// TIA Portal project "Semafoare_2026" (V15.1)

(* hardware
DEVICE "S71500/ET200MP station_1"  S7-1500 station
   slot 0: "Rail_0"  Rack  6ES7 590-1***0-0AA0
   slot 1: "PLC_1"  CPU 1513-1 PN  6ES7 513-1AL02-0AB0  V2.6
      slot 3: "CPU display_1"  6ES7591-1AA00-0AA0
DEVICE "HMI_1"  KTP900 Basic PN
   slot 0: "HMI_1"  KTP900 Basic PN  6AV2 123-2JB03-0AX0  15.1.0.0
   slot 1: "HMI_RT_1"  KTP900 Basic PN  6AV2 123-2JB03-0AX0  15.1.0.0
   slot 5: "HMI_1.IE_CP_1"  PROFINET Interface  15.0.1.0
      slot 1: "PROFINET Interface_1"  PROFINET Interface
         slot 1: "Port_1"  Port
*)

// ===== PLC "PLC_1"  CPU 1513-1 PN =====

VAR_GLOBAL   // PLC tag table "Default tag table"
   "Clock_Byte" AT %MB0 : Byte;
   "Clock_10Hz" AT %M0.0 : Bool;
   "Clock_5Hz" AT %M0.1 : Bool;
   "Clock_2.5Hz" AT %M0.2 : Bool;
   "Clock_2Hz" AT %M0.3 : Bool;
   "Clock_1.25Hz" AT %M0.4 : Bool;
   "Clock_1Hz" AT %M0.5 : Bool;
   "Clock_0.625Hz" AT %M0.6 : Bool;
   "Clock_0.5Hz" AT %M0.7 : Bool;
END_VAR

DATA_BLOCK "Semafor_masini_ciclu_DB"   // DB1
{ S7_Optimized_Access := 'TRUE' }
VERSION : 0.1
   VAR
      rosu_on : Bool;
      galben_on : Bool;
      galben_on_hmi : Bool;
      verde_on : Bool;
      time_elapsed_rosu : Time;
      time_elapsed_rosu_secunde : Time;
      time_elapsed_verde : Time;
      time_elapsed_verde_secunde : Time;
      time_elapsed_galben : Time;
      time_elapsed_galben_secunde : Time;
      "mod" : Int;
   END_VAR
BEGIN
END_DATA_BLOCK

DATA_BLOCK "Semafor_pietoni_DB"   // DB2
{ S7_Optimized_Access := 'TRUE' }
VERSION : 0.1
BEGIN
END_DATA_BLOCK

DATA_BLOCK "Semafor_masini_ciclu_DB_1"   // DB3
{ S7_Optimized_Access := 'TRUE' }
VERSION : 0.1
// stored: InstanceOfName Semafor_masini_ciclu
"Semafor_masini_ciclu"
BEGIN
END_DATA_BLOCK

FUNCTION_BLOCK "Semafor_masini_ciclu"   // FB1, LAD
{ S7_Optimized_Access := 'TRUE' }
VERSION : 0.1
   VAR_INPUT
      mod_functinare : Int;
   END_VAR
   VAR_OUTPUT
      time_elapsed_verde : Time;
      time_elapsed_galben : Time;
      time_elapsed_rosu : Time;
   END_VAR
   VAR_IN_OUT
      verde_on : Bool;
      rosu_on : Bool;
      galben_on : Bool;
   END_VAR
   VAR
      timer_rosu : TON_TIME;
      timer_galben : TON_TIME;
      timer_verde : TON_TIME;
      galben_intermitent_on : Bool;
      re1 : Bool;
      re_aux : Bool;
      mod_normal : Bool;
      reseteaza_ciclul : Bool;
      porneste_verde : Bool;
      porneste_rosu : Bool;
      porneste_galben : Bool;
   END_VAR
   VAR_TEMP   // added for the SCL form of the ladder/FBD networks
      _w1 : Bool;
   END_VAR
BEGIN

REGION Network 1: semafor modul normal/mod oprire
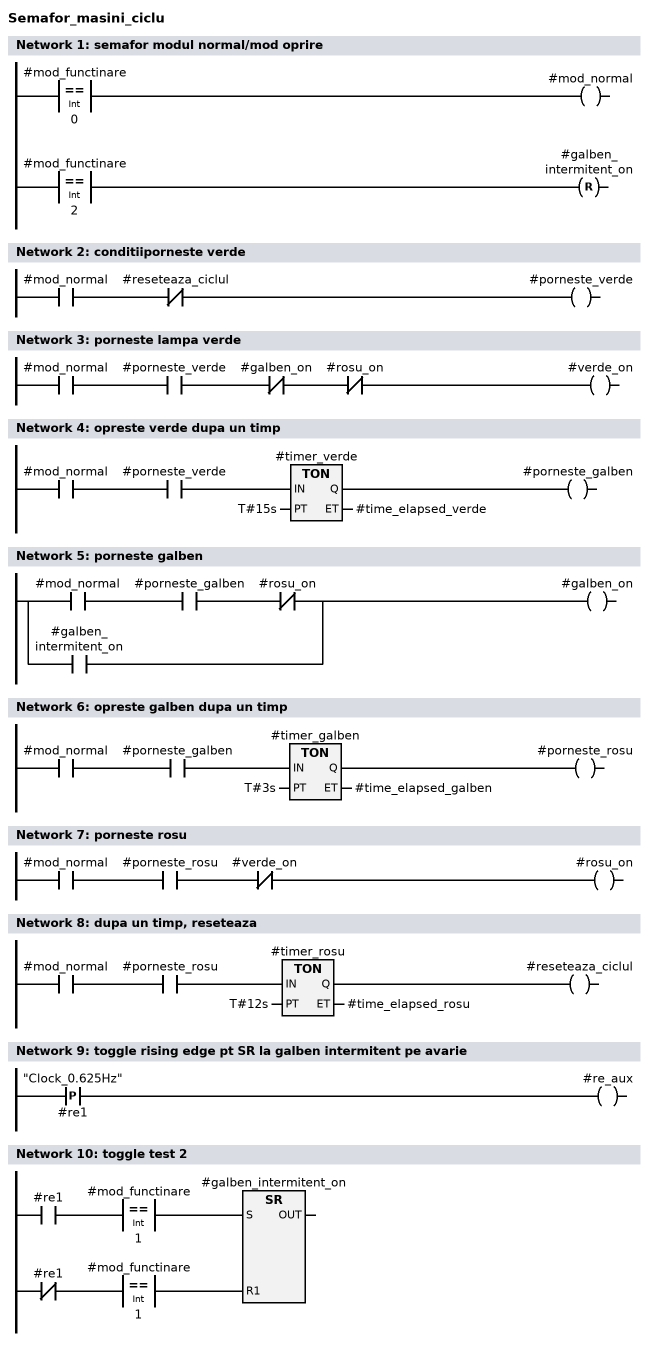
   RUNG wire#powerrail
      { S7_Templates := "SrcType := Int" } EQ_Contact(in1 := #mod_functinare, in2 := 0)
      Coil( #mod_normal )
   END_RUNG
   RUNG wire#powerrail
      { S7_Templates := "SrcType := Int" } EQ_Contact(in1 := #mod_functinare, in2 := 2)
      R_Coil( #galben_intermitent_on )
   END_RUNG
   // the same network as SCL:
   #mod_normal := #mod_functinare = 0;
   IF #mod_functinare = 2 THEN #galben_intermitent_on := FALSE; END_IF;
END_REGION

REGION Network 2: conditiiporneste verde
   RUNG wire#powerrail
      Contact( #mod_normal )
      I_Contact( #reseteaza_ciclul )
      Coil( #porneste_verde )
   END_RUNG
   // the same network as SCL:
   #porneste_verde := #mod_normal AND NOT #reseteaza_ciclul;
END_REGION

REGION Network 3: porneste lampa verde
   RUNG wire#powerrail
      Contact( #mod_normal )
      Contact( #porneste_verde )
      I_Contact( #galben_on )
      I_Contact( #rosu_on )
      Coil( #verde_on )
   END_RUNG
   // the same network as SCL:
   #verde_on := #mod_normal AND #porneste_verde AND NOT #galben_on AND NOT #rosu_on;
END_REGION

REGION Network 4: opreste verde dupa un timp
   #timer_verde(IN := #mod_normal AND #porneste_verde, PT := T#15s, ET => #time_elapsed_verde);   // TON
   #porneste_galben := #timer_verde.Q;
END_REGION

REGION Network 5: porneste galben
   RUNG wire#powerrail
      Contact( #mod_normal )
      Contact( #porneste_galben )
      I_Contact( #rosu_on )
      wire#w1
      Coil( #galben_on )
   END_RUNG
   RUNG wire#powerrail
      Contact( #galben_intermitent_on )
   END_RUNG wire#w1
   // the same network as SCL:
   #galben_on := (#mod_normal AND #porneste_galben AND NOT #rosu_on) OR #galben_intermitent_on;
END_REGION

REGION Network 6: opreste galben dupa un timp
   #timer_galben(IN := #mod_normal AND #porneste_galben, PT := T#3s, ET => #time_elapsed_galben);   // TON
   #porneste_rosu := #timer_galben.Q;
END_REGION

REGION Network 7: porneste rosu
   RUNG wire#powerrail
      Contact( #mod_normal )
      Contact( #porneste_rosu )
      I_Contact( #verde_on )
      Coil( #rosu_on )
   END_RUNG
   // the same network as SCL:
   #rosu_on := #mod_normal AND #porneste_rosu AND NOT #verde_on;
END_REGION

REGION Network 8: dupa un timp, reseteaza
   #timer_rosu(IN := #mod_normal AND #porneste_rosu, PT := T#12s, ET => #time_elapsed_rosu);   // TON
   #reseteaza_ciclul := #timer_rosu.Q;
END_REGION

REGION Network 9: toggle rising edge pt SR la galben intermitent pe avarie
   RUNG wire#powerrail
      P_Contact(operand := "Clock_0.625Hz", bit := #re1)
      Coil( #re_aux )
   END_RUNG
   // the same network as SCL:
   #_w1 := "Clock_0.625Hz" AND NOT #re1;   // rising edge of "Clock_0.625Hz"
   #re1 := "Clock_0.625Hz";
   #re_aux := #_w1;
END_REGION

REGION Network 10: toggle test 2
   RUNG wire#powerrail
      Contact( #re1 )
      { S7_Templates := "SrcType := Int" } EQ_Contact(in1 := #mod_functinare, in2 := 1)
      S_SR(operand := #galben_intermitent_on, r1 := wire#w1)
   END_RUNG
   RUNG wire#powerrail
      I_Contact( #re1 )
      { S7_Templates := "SrcType := Int" } EQ_Contact(in1 := #mod_functinare, in2 := 1)
   END_RUNG wire#w1
   // the same network as SCL:
   IF #re1 AND (#mod_functinare = 1) THEN
       #galben_intermitent_on := TRUE;   // SR flip-flop
   END_IF;
   IF NOT #re1 AND (#mod_functinare = 1) THEN #galben_intermitent_on := FALSE; END_IF;
END_REGION
END_FUNCTION_BLOCK

FUNCTION_BLOCK "Semafor_pietoni"   // FB2, LAD
{ S7_Optimized_Access := 'TRUE' }
VERSION : 0.1
BEGIN
END_FUNCTION_BLOCK

ORGANIZATION_BLOCK "Main"   // OB1, LAD, ProgramCycle
TITLE = "Main Program Sweep (Cycle)"
{ S7_Optimized_Access := 'TRUE' }
VERSION : 0.1
   VAR_INPUT
      Initial_Call : Bool;   // Initial call of this OB
      Remanence : Bool;   // =True, if remanent data are available
   END_VAR
BEGIN

REGION Network 1: Semafor masini ciclu
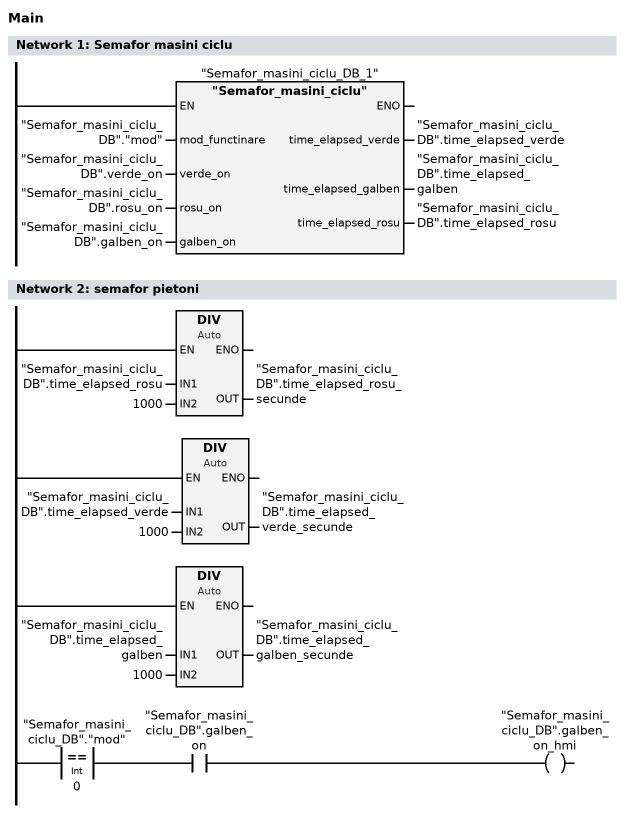
   RUNG wire#powerrail
      "Semafor_masini_ciclu_DB_1"(mod_functinare := "Semafor_masini_ciclu_DB"."mod", verde_on := "Semafor_masini_ciclu_DB".verde_on, rosu_on := "Semafor_masini_ciclu_DB".rosu_on, galben_on := "Semafor_masini_ciclu_DB".galben_on, time_elapsed_verde => "Semafor_masini_ciclu_DB".time_elapsed_verde, time_elapsed_galben => "Semafor_masini_ciclu_DB".time_elapsed_galben, time_elapsed_rosu => "Semafor_masini_ciclu_DB".time_elapsed_rosu)
   END_RUNG
   // the same network as SCL:
   "Semafor_masini_ciclu_DB_1"(mod_functinare := "Semafor_masini_ciclu_DB"."mod",   // "Semafor_masini_ciclu"
                           verde_on := "Semafor_masini_ciclu_DB".verde_on,
                           rosu_on := "Semafor_masini_ciclu_DB".rosu_on,
                           galben_on := "Semafor_masini_ciclu_DB".galben_on,
                           time_elapsed_verde => "Semafor_masini_ciclu_DB".time_elapsed_verde,
                           time_elapsed_galben => "Semafor_masini_ciclu_DB".time_elapsed_galben,
                           time_elapsed_rosu => "Semafor_masini_ciclu_DB".time_elapsed_rosu);
END_REGION

REGION Network 2: semafor pietoni
   RUNG wire#powerrail
      Div(in1 := "Semafor_masini_ciclu_DB".time_elapsed_rosu, in2 := 1000, out => "Semafor_masini_ciclu_DB".time_elapsed_rosu_secunde)
   END_RUNG
   RUNG wire#powerrail
      Div(in1 := "Semafor_masini_ciclu_DB".time_elapsed_verde, in2 := 1000, out => "Semafor_masini_ciclu_DB".time_elapsed_verde_secunde)
   END_RUNG
   RUNG wire#powerrail
      Div(in1 := "Semafor_masini_ciclu_DB".time_elapsed_galben, in2 := 1000, out => "Semafor_masini_ciclu_DB".time_elapsed_galben_secunde)
   END_RUNG
   RUNG wire#powerrail
      { S7_Templates := "SrcType := Int" } EQ_Contact(in1 := "Semafor_masini_ciclu_DB"."mod", in2 := 0)
      Contact( "Semafor_masini_ciclu_DB".galben_on )
      Coil( "Semafor_masini_ciclu_DB".galben_on_hmi )
   END_RUNG
   // the same network as SCL:
   "Semafor_masini_ciclu_DB".time_elapsed_rosu_secunde := "Semafor_masini_ciclu_DB".time_elapsed_rosu / 1000;
   "Semafor_masini_ciclu_DB".time_elapsed_verde_secunde := "Semafor_masini_ciclu_DB".time_elapsed_verde / 1000;
   "Semafor_masini_ciclu_DB".time_elapsed_galben_secunde := "Semafor_masini_ciclu_DB".time_elapsed_galben / 1000;
   "Semafor_masini_ciclu_DB".galben_on_hmi := ("Semafor_masini_ciclu_DB"."mod" = 0) AND "Semafor_masini_ciclu_DB".galben_on;
END_REGION

REGION Network 3: timp in secunde
END_REGION
END_ORGANIZATION_BLOCK

(* ===== HMI "HMI_RT_1" =====
system functions are stored by id; their names below are inferred from use
connection "HMI_Connection_1": ETHERNET, SMART_S7_1500_OMS

HMI tags "Default tag table"
   "Semafor_masini_ciclu_DB_rosu_on" : Bool = PLC Semafor_masini_ciclu_DB.rosu_on, 1 s
   "Semafor_masini_ciclu_DB_galben_on" : Bool = PLC Semafor_masini_ciclu_DB.galben_on AT %DB1.DBX0.0, 1 s
   "Semafor_masini_ciclu_DB_verde_on" : Bool = PLC Semafor_masini_ciclu_DB.verde_on AT %DB1.DBX0.0, 1 s
   "Semafor_masini_ciclu_DB_mod" : Int = PLC Semafor_masini_ciclu_DB.mod AT %DB1.DBX0.0, 1 s
   "Semafor_masini_ciclu_DB_time_elapsed_rosu_secunde" : Time = PLC Semafor_masini_ciclu_DB.time_elapsed_rosu_secunde, 1 s
   "Semafor_masini_ciclu_DB_time_elapsed_verde_secunde" : Time = PLC Semafor_masini_ciclu_DB.time_elapsed_verde_secunde, 1 s
   "Semafor_masini_ciclu_DB_time_elapsed_galben_secunde" : Time = PLC Semafor_masini_ciclu_DB.time_elapsed_galben_secunde, 1 s
   "Semafor_masini_ciclu_DB_galben_on_hmi" : Bool = PLC Semafor_masini_ciclu_DB.galben_on_hmi, 1 s

Template "Template_1" 800x480
   Button "Exit" at 722,440 size 55x39; TextOff 'Exit'; PictureOff "ExitRuntime_KTP900_Basic_PN_TR"; PictureOn "ExitRuntime_KTP900_Basic_PN_TR"
      on Release: StopRuntime(0)

screen "Semafor_ciclu" 800x480, template "Template_1"
   Circle "Circle_1" at 390,53 size 44x44
      Appearance <- "Semafor_masini_ciclu_DB_rosu_on"
   Circle "Circle_2" at 390,115 size 44x44
      Appearance <- "Semafor_masini_ciclu_DB_galben_on"
   Circle "Circle_3" at 390,178 size 44x44
      Appearance <- "Semafor_masini_ciclu_DB_verde_on"
   Button "Button_1" at 121,86 size 84x32; TextOff 'Pornire'
      on Activate: SetTag("Semafor_masini_ciclu_DB_mod", 0)
      Appearance <- "Semafor_masini_ciclu_DB_mod"
   Button "Button_2" at 121,127 size 84x32; TextOff 'Oprire'
      on Activate: SetTag("Semafor_masini_ciclu_DB_mod", 2)
      Appearance <- "Semafor_masini_ciclu_DB_mod"
   Button "Button_3" at 121,168 size 84x32; TextOff 'Intermitent'
      on Activate: SetTag("Semafor_masini_ciclu_DB_mod", 1)
      Appearance <- "Semafor_masini_ciclu_DB_mod"
   IOField "I/O field_1" at 495,54 size 96x32; FormatPattern 999; Unit s
      ProcessValue <- "Semafor_masini_ciclu_DB_time_elapsed_rosu_secunde"
      Visibility <- "Semafor_masini_ciclu_DB_rosu_on"
   IOField "I/O field_2" at 495,190 size 96x32; FormatPattern 999; Unit s
      ProcessValue <- "Semafor_masini_ciclu_DB_time_elapsed_verde_secunde"
      Visibility <- "Semafor_masini_ciclu_DB_verde_on"
   IOField "I/O field_3" at 495,120 size 96x32; FormatPattern 999; Unit s
      ProcessValue <- "Semafor_masini_ciclu_DB_time_elapsed_galben_secunde"
      Visibility <- "Semafor_masini_ciclu_DB_galben_on_hmi"
*)